PROGRAM MAIN
VAR
END_VAR

GVL_HMI.hmiPanel();

UpperPreserDrive();
HydraulicPump();
BreakthroughDetection_2();



P_Events();
P_EventsDefinition();
Alarms();
Scaling();
SavePresistent();
Mode();
IO_Map();

END_PROGRAM

(* stored: Version 1.1.0.1, ProductVersion 3.1.4024.15
   POU MAIN: Id {93197c60-806b-4e15-b6d1-f529f30b5b27}, SpecialFunc None *)
